Fanuc KAREL source: NC0086.KL

-- PROVISIONAL review KL for V1013-1; original PC SHA256 446f40c759a69ce51538d50747659ae052bdad54e40d8ca5380be7de72c66096
-- Incomplete behavior may be omitted. Consult companion uncertainty JSON. Do not deploy.
PROGRAM NC0086
%NOLOCKGROUP
-- UNRESOLVED_LOCAL_POOL 3 cells at code offset 3; source declarations unknown
-- DIRECT_LOCAL_WORD_ACCESS alone does not prove INTEGER, REAL, or BOOLEAN
BEGIN
  -- UNRESOLVED_PC offsets 0-8; opcodes 2B,2C,7B
  -- UNRESOLVED_PC offsets 13-20; opcodes 9D,23
  -- UNRESOLVED_PC offsets 25-38; opcodes 21,9D,57,79
  -- UNRESOLVED_PC offsets 43-60; opcodes 21,40,41,42
  -- UNRESOLVED_PC offsets 65-94; opcodes 9D,23,9E,2E,22,7A
  -- UNRESOLVED_PC offsets 99-116; opcodes 21,2E,59,79
  -- UNRESOLVED_PC offsets 121-134; opcodes 21,9D,57,79
  -- UNRESOLVED_PC offsets 139-156; opcodes 21,40,41,42
  -- UNRESOLVED_PC offsets 161-190; opcodes 9D,23,9E,2E,22,7A
  -- UNRESOLVED_PC offsets 195-212; opcodes 21,2E,59,79
  -- UNRESOLVED_PC offsets 217-231; opcodes 21,9D,52,23
  -- UNRESOLVED_PC offsets 236-241; opcodes 7A
  -- UNRESOLVED_PC offsets 246-277; opcodes 20,2C,23,7A,40,41,42
  -- UNRESOLVED_PC offsets 282-306; opcodes 21,2E,52,23,7A,43
  -- UNRESOLVED_PC offsets 311-329; opcodes 21,2E,52,23
  -- UNRESOLVED_PC offsets 339-344; opcodes 7A
  -- UNRESOLVED_PC offsets 349-367; opcodes 21,2E,52,23
  -- UNRESOLVED_PC offsets 377-382; opcodes 7A
  -- UNRESOLVED_PC offsets 387-418; opcodes 20,2C,23,7A,40,41,42
  -- UNRESOLVED_PC offsets 423-447; opcodes 21,2E,52,23,7A,43
  -- UNRESOLVED_PC offsets 452-470; opcodes 21,2E,52,23
  -- UNRESOLVED_PC offsets 480-485; opcodes 7A
  -- UNRESOLVED_PC offsets 490-508; opcodes 21,2E,52,23
  -- UNRESOLVED_PC offsets 518-522; opcodes 7F
  -- UNRESOLVED_PC offsets 527-531; opcodes 27,AA
  -- UNRESOLVED_PC offsets 536-540; opcodes 7F
END NC0086
